{attribute 'OPC.UA.DA.StructuredType' := '1'}
TYPE ST_HeatPumpState :
STRUCT
	bError					: BOOL;
END_STRUCT
END_TYPE

(* stored: Version 1.1.0.1, ProductVersion 3.1.4024.10
   DUT ST_HeatPumpState: Id {24917478-f4f3-4529-90c5-06421d5b907a} *)
